// TIA Portal V19 export
FUNCTION_BLOCK "TYPIC_C501_IF_BBP"   // FB19, FBD
TITLE = TYPIC_C501_IF_BBP: Brandbluspomp
{ S7_Optimized_Access := 'TRUE' }
AUTHOR : OCOTECH
FAMILY : Typical
NAME : C501.707
// Logisch Object Besturing: C501.707
// 
// De interne functie brandbluspomp verzorgt de interne besturing, bewaking en fysieke aansturing van een brandbluspomp behorend tot de brandblusinstallatie.
// stored: MemoryReserve 10, SetENOAutomatically false
   VAR_INPUT
      PULS_100ms { ExternalAccessible := 'False'; ExternalVisible := 'False'; ExternalWritable := 'False'} : Bool;   // Puls, 1 PLC-cyclus hoog, 1 keer per 100 ms
      PULS_1s { ExternalAccessible := 'False'; ExternalVisible := 'False'; ExternalWritable := 'False'} : Bool;   // Puls, 1 PLC-cyclus hoog, 1 keer per seconde
      EXT_HW { ExternalAccessible := 'False'; ExternalVisible := 'False'; ExternalWritable := 'False'} : Bool;   // Sturings hardware (PLC) bewaking (1 = OK)
      IN_HND { ExternalAccessible := 'False'; ExternalVisible := 'False'; ExternalWritable := 'False'} : Bool;   // Terugmelding aansturing via hand (hardware)
      IN_AAN { ExternalAccessible := 'False'; ExternalVisible := 'False'; ExternalWritable := 'False'} : Bool;   // Terugmelding aansturing
      IN_AUT_C501 { ExternalAccessible := 'False'; ExternalVisible := 'False'; ExternalWritable := 'False'} : Bool;   // Beveiligingen: serie geschakelde terugmelding (1= OK)
      IN_AUT { ExternalAccessible := 'False'; ExternalVisible := 'False'; ExternalWritable := 'False'} : Bool;   // Status thermische beveiliging (1 = OK)
      IN_PTC { ExternalAccessible := 'False'; ExternalVisible := 'False'; ExternalWritable := 'False'} : Bool;   // Detectie hoge temperatuur in de wikkelingen van de motor (1 = OK)
      IN_SCW { ExternalAccessible := 'False'; ExternalVisible := 'False'; ExternalWritable := 'False'} : Bool;   // Werkschakelaar (1 = Aan)
      IN_STO { ExternalAccessible := 'False'; ExternalVisible := 'False'; ExternalWritable := 'False'} : Bool;   // Status Softstarter (1 = OK)
      IN_DME_STO { ExternalAccessible := 'False'; ExternalVisible := 'False'; ExternalWritable := 'False'} : Bool;   // Filterbewaking (1= OK / 0 = Vervuild)
      IN_STS1 { ExternalAccessible := 'False'; ExternalVisible := 'False'; ExternalWritable := 'False'} : Bool;   // Status motorlade ingeschakeld
      IN_STS2 { ExternalAccessible := 'False'; ExternalVisible := 'False'; ExternalWritable := 'False'} : Bool;   // Status motorlade in test
      IN_STS3 { ExternalAccessible := 'False'; ExternalVisible := 'False'; ExternalWritable := 'False'} : Bool;   // Status motorlade uitgereden
      IN_STR1 { ExternalAccessible := 'False'; ExternalVisible := 'False'; ExternalWritable := 'False'} : Int;   // Analoge meting ventilator fasestroom 1
      IN_STR2 { ExternalAccessible := 'False'; ExternalVisible := 'False'; ExternalWritable := 'False'} : Int;   // Analoge meting ventilator fasestroom 2
      IN_STR3 { ExternalAccessible := 'False'; ExternalVisible := 'False'; ExternalWritable := 'False'} : Int;   // Analoge meting ventilator fasestroom 3
      IN_TRL { ExternalAccessible := 'False'; ExternalVisible := 'False'; ExternalWritable := 'False'} : Bool;   // Trillingsdetectie (1 = Geen trillingen)
      CFG_TYD_FB { ExternalAccessible := 'False'; ExternalVisible := 'False'; ExternalWritable := 'False'} : Time;   // Vertragingstijd storing foute terugmelding
      CFG_TYD_TRL { ExternalAccessible := 'False'; ExternalVisible := 'False'; ExternalWritable := 'False'} : Time;   // Vertragingstijd storing onbalans
      CFG_TRL_MAX { ExternalAccessible := 'False'; ExternalVisible := 'False'; ExternalWritable := 'False'} : Real;   // Hoogste waarde scalering trillingsmeting
      CFG_TRL_MIN { ExternalAccessible := 'False'; ExternalVisible := 'False'; ExternalWritable := 'False'} : Real;   // Laagste waarde scalering trillingsmeting
      CFG_TRL_HOOG { ExternalAccessible := 'False'; ExternalVisible := 'False'; ExternalWritable := 'False'} : Real;   // Schakeldrempel hoog trillingsmeting (onbalans)
      CFG_TYD_RUN { ExternalAccessible := 'False'; ExternalVisible := 'False'; ExternalWritable := 'False'} : LInt;   // Minimale draaitijd om melding onderhoud nodig te resetten
      CFG_TYD_STOP { ExternalAccessible := 'False'; ExternalVisible := 'False'; ExternalWritable := 'False'} : LInt;   // Stilstandstijd die melding onderhoud nodig activeert
      CFG_TYD_MAX { ExternalAccessible := 'False'; ExternalVisible := 'False'; ExternalWritable := 'False'} : Int;   // Tijdsduur draaitijd overschrijding pomp
   END_VAR
   VAR_OUTPUT
      VAR_IF_BBP { ExternalAccessible := 'False'; ExternalVisible := 'False'; ExternalWritable := 'False'} : "C501_VAR_IF_BBP_TYPIC";   // Struct met alle variabelen naar bovenliggende functies
      OUT_AAN { ExternalAccessible := 'False'; ExternalVisible := 'False'; ExternalWritable := 'False'} : Bool;   // Aansturen pomp
      OUT_RES { ExternalAccessible := 'False'; ExternalVisible := 'False'; ExternalWritable := 'False'} : Bool;   // Reset softstarter
   END_VAR
   VAR_IN_OUT
      STU_IF_BBP : "C501_STU_IF_BBP_TYPIC";   // Struct met alle sturingen van de subfunctie (SF) pomp van 3B
   END_VAR
   VAR
      BED : Struct   // Bedieningen
         REM : Bool;   // Bediening om pomp in Remote te schakelen (indien IN_HND = 0)
         FWD : Bool;   // Bediening om pomp in hand te schakelen en te starten
         STOP : Bool;   // Bediening om pomp in hand te schakelen en te stoppen
         RES : Bool;   // Reset storingen
      END_STRUCT;
      STO { ExternalWritable := 'False'} : Struct   // Storingen
         A001 : Bool;   // Beveiliging aangesproken
         A002 : Bool;   // Storing van de motorbeveiliging van de pomp
         A003 : Bool;   // Storing softstarter
         A004 : Bool;   // Te hoge temperatuur in de motorwikkelingen
         A005 : Bool;   // De pomp is in onbalans
         A006 : Bool;   // Motorlade uitgeschakeld
         A007 : Bool;   // Motorlade in test
         A008 : Bool;   // Motorlade uitgereden
         A009 : Bool;   // Fout stroommeting fase 1
         A010 : Bool;   // Fout stroommeting fase 2
         A011 : Bool;   // Fout stroommeting fase 3
         A012 : Bool;   // Filter vervuild
         AT01 : Bool;   // Discordantie motor: terugmelding niet ontvangen
         AT02 : Bool;   // Discordantie motor: terugmelding blijft aanwezig
         M001 : Bool;   // Werkschakelaar uitgeschakeld
         M002 : Bool;   // Melding: Pomp heeft te lang niet gedraaid. Periodiek onderhoud nodig
         M003 : Bool;   // Melding: Draaitijd overschrijding
      END_STRUCT;
      VAR { ExternalWritable := 'False'} : Struct   // Variabelen
         STS_AAN : Bool;   // Pomp draait
         BMO_HAND : Bool;   // Pomp in hand geschakeld
         TYD_TOT_AAN { ExternalAccessible := 'False'; ExternalVisible := 'False'} : LInt;   // Totaal aantal draaiuren (in seconden)
         TYD_TOT_AAN_UUR { ExternalAccessible := 'False'; ExternalVisible := 'False'} : LInt;   // Totaal aantal draaiuren (in uren)
         TYD_AAN { ExternalAccessible := 'False'; ExternalVisible := 'False'} : Int;   // Aantal seconden dat pomp aangeschakeld is
         TYD_UIT { ExternalAccessible := 'False'; ExternalVisible := 'False'} : Int;   // Aantal seconden dat pomp uitgeschakeld is
         ENE_MWA1 { ExternalAccessible := 'False'; ExternalVisible := 'False'} : Real;   // Stroommeting fase 1
         ENE_MWA2 { ExternalAccessible := 'False'; ExternalVisible := 'False'} : Real;   // Stroommeting fase 2
         ENE_MWA3 { ExternalAccessible := 'False'; ExternalVisible := 'False'} : Real;   // Stroommeting fase 3
         EXT_HW { ExternalAccessible := 'False'; ExternalVisible := 'False'} : Bool;   // Sturings hardware (PLC) in storing
      END_STRUCT;
   END_VAR
BEGIN

REGION Network 1: START
END_REGION

REGION Network 2: +++ Metingen +++
   // Inlezen van de 3 stroommetingen van iedere fase van de motor.
END_REGION

REGION Network 3: +++ Storingen +++
   // Verwerken van de storingsmeldingen (inputs).
END_REGION

REGION Network 4: Storing A001: Beveiliging aangesproken
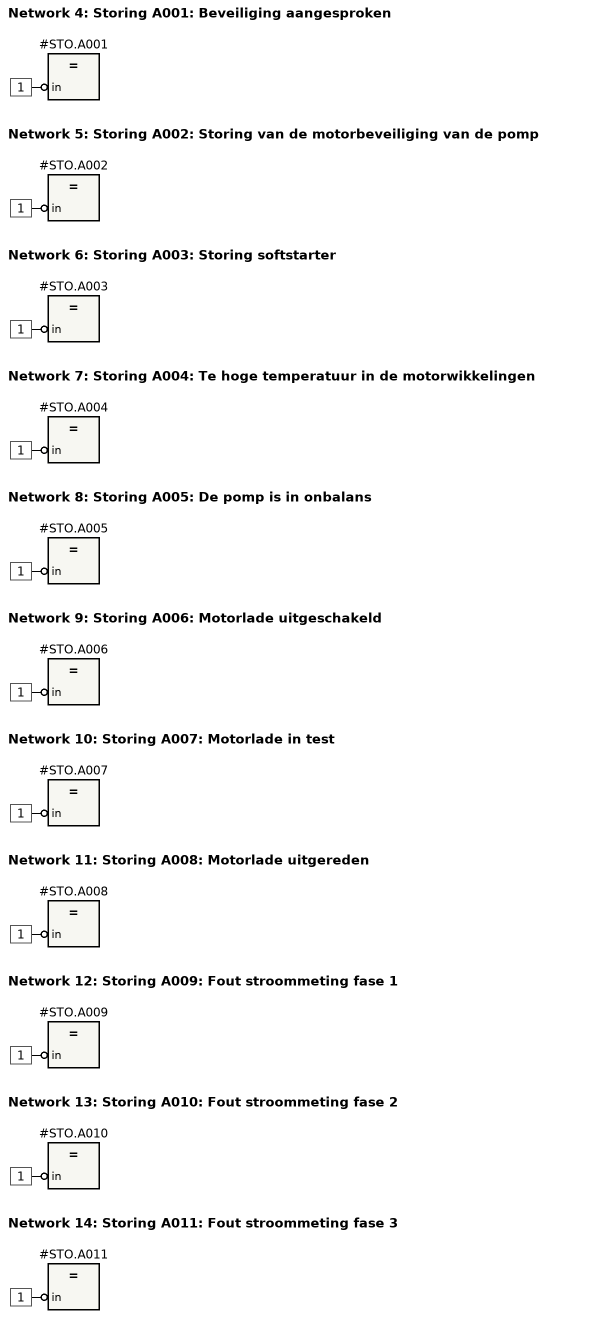
   #STO.A001 := NOT 1;
END_REGION

REGION Network 5: Storing A002: Storing van de motorbeveiliging van de pomp
   #STO.A002 := NOT 1;
END_REGION

REGION Network 6: Storing A003: Storing softstarter
   #STO.A003 := NOT 1;
END_REGION

REGION Network 7: Storing A004: Te hoge temperatuur in de motorwikkelingen
   #STO.A004 := NOT 1;
END_REGION

REGION Network 8: Storing A005: De pomp is in onbalans
   #STO.A005 := NOT 1;
END_REGION

REGION Network 9: Storing A006: Motorlade uitgeschakeld
   #STO.A006 := NOT 1;
END_REGION

REGION Network 10: Storing A007: Motorlade in test
   #STO.A007 := NOT 1;
END_REGION

REGION Network 11: Storing A008: Motorlade uitgereden
   #STO.A008 := NOT 1;
END_REGION

REGION Network 12: Storing A009: Fout stroommeting fase 1
   #STO.A009 := NOT 1;
END_REGION

REGION Network 13: Storing A010: Fout stroommeting fase 2
   #STO.A010 := NOT 1;
END_REGION

REGION Network 14: Storing A011: Fout stroommeting fase 3
   #STO.A011 := NOT 1;
END_REGION

REGION Network 15: Storing A012: Filter vervuild
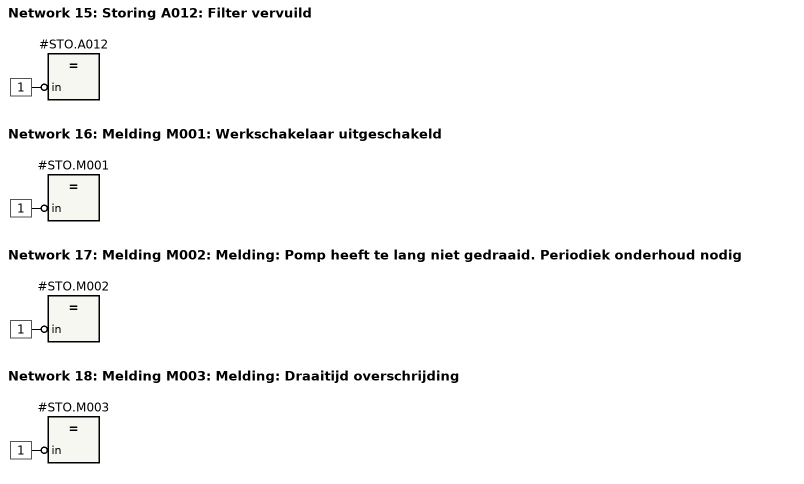
   #STO.A012 := NOT 1;
END_REGION

REGION Network 16: Melding M001: Werkschakelaar uitgeschakeld
   #STO.M001 := NOT 1;
END_REGION

REGION Network 17: Melding M002: Melding: Pomp heeft te lang niet gedraaid. Periodiek onderhoud nodig
   #STO.M002 := NOT 1;
END_REGION

REGION Network 18: Melding M003: Melding: Draaitijd overschrijding
   #STO.M003 := NOT 1;
END_REGION

REGION Network 19: +++ Motorsturing +++
   // Aansturen en bewaking van de motor.
END_REGION

REGION Network 20: +++ Urentellers +++
   // Tellen van de tijdsduur dat motor draait of stilstaat.
END_REGION

REGION Network 21 (SCL): EINDE
   // Variabelen van intern scada rakvlak naar outputs copieren
   #VAR_IF_BBP.STS_AAN := #VAR.STS_AAN;
   #VAR_IF_BBP.BMO_HAND := #VAR.BMO_HAND;
   #VAR_IF_BBP.TYD_TOT_AAN := #VAR.TYD_TOT_AAN;
   #VAR_IF_BBP.TYD_TOT_AAN_UUR := #VAR.TYD_TOT_AAN_UUR;
   #VAR_IF_BBP.TYD_AAN := #VAR.TYD_AAN;
   #VAR_IF_BBP.TYD_UIT := #VAR.TYD_UIT;
   #VAR_IF_BBP.ENE_MWA1 := #VAR.ENE_MWA1;
   #VAR_IF_BBP.ENE_MWA2 := #VAR.ENE_MWA2;
   #VAR_IF_BBP.ENE_MWA3 := #VAR.ENE_MWA3;
   #VAR_IF_BBP.EXT_HW := #VAR.EXT_HW;
   #VAR_IF_BBP.STO := #STO;
END_REGION
END_FUNCTION_BLOCK
